// TIA Portal V20 export
TYPE "LKinCtrl_typePathData"
   STRUCT
      pathDataName : String["LKINCTRL_LENGTH_OF_PATHDATA_NAME"];   // name of PathData
      LKinLangInterface : "LKinCtrl_typeAdvPointers";   // pointers to add / retrieve cmds in PathData
      commands : Array[1.."LKINCTRL_NO_OF_PATHDATA_ELEMENTS"] of "LKinCtrl_typePathDataElement";   // command list
   END_STRUCT;
   // commands[1].cmdParameters.transitionParameters[1] := -1.0;
   // commands[2].cmdParameters.transitionParameters[1] := -1.0;
   // commands[3].cmdParameters.transitionParameters[1] := -1.0;
   // commands[4].cmdParameters.transitionParameters[1] := -1.0;
   // commands[5].cmdParameters.transitionParameters[1] := -1.0;
   // commands[6].cmdParameters.transitionParameters[1] := -1.0;
   // commands[7].cmdParameters.transitionParameters[1] := -1.0;
   // commands[8].cmdParameters.transitionParameters[1] := -1.0;
   // commands[9].cmdParameters.transitionParameters[1] := -1.0;
   // commands[10].cmdParameters.transitionParameters[1] := -1.0;
   // commands[11].cmdParameters.transitionParameters[1] := -1.0;
   // commands[12].cmdParameters.transitionParameters[1] := -1.0;
   // commands[13].cmdParameters.transitionParameters[1] := -1.0;
   // commands[14].cmdParameters.transitionParameters[1] := -1.0;
   // commands[15].cmdParameters.transitionParameters[1] := -1.0;
   // commands[16].cmdParameters.transitionParameters[1] := -1.0;
   // commands[17].cmdParameters.transitionParameters[1] := -1.0;
   // commands[18].cmdParameters.transitionParameters[1] := -1.0;
   // commands[19].cmdParameters.transitionParameters[1] := -1.0;
   // commands[20].cmdParameters.transitionParameters[1] := -1.0;
END_TYPE
